(* PLC project CoDeSys External Library Template, WAGO e!COCKPIT e!COCKPIT, author 3S - Smart Software Solutions GmbH *)
(* stored: creationDateTime 2019-10-29T12:22:40.3974988, version 3.5.5.30, modificationDateTime 2019-10-24T14:40:07.960949, organization 3S - Smart Software Solutions GmbH *)
(* Library project template with all possible element types, docu and a sample project structure *)

(* values of enumPPPSKlimatyzatorTroxSchoolairVError: BrakKomunikacji: brak komunikacji z węzłem; AlarmCzujnika: alarm braku zmiany wartości czujnika temp. *)

(* Autor: Artur Wyszomirski, 2019-02-05-AWy Prawa majątkowe: Solwena Sp. z o.o., Aktualizacje: 2019-02-18-AWy - alarm czujnika temperatury Opis: enum służy do obsługi alarmów w fb węzła Frisko ATTOM1S na budynkach PPP Sopot (ENGIE) *)
{attribute 'qualified_only'}
{attribute 'strict'}
TYPE enumPPPSKlimatyzatorTroxSchoolairVError : (BrakKomunikacji := 1, AlarmCzujnika := 2);
END_TYPE
